Omron CX-Programmer project NewProject (CX-Programmer 9.50)

# PLC NewPLC1: CJ2M CPU35
I/O table (CPU CJ2M-CPU35): rack 0 slot 0 CJ1W-SCU41-V1; rack 0 slot 1 CJ1W-ID211; rack 0 slot 2 CJ1W-ID211; rack 0 slot 3 CJ1W-OC211; rack 0 slot 11 CJ2M-EIP21

## Global symbols (name address type ; comment)
0.00 BOOL  ; st
0.01 BOOL  ; sensor1
0.03 BOOL  ; metal detector
0.05 BOOL  ; sensor3
0.07 BOOL  ; sensor C4_R
0.09 BOOL  ; sensor C4_F
1.01 BOOL  ; sensor1
1.03 BOOL  ; SensorB2
1.05 BOOL  ; sensorP2_3
20.00 BOOL  ; st
20.01 BOOL  ; CR2
2.00 BOOL  ; e
2.01 BOOL  ; CR1
2.02 BOOL  ; pin28
2.03 BOOL  ; pin30
2.04 BOOL  ; pin36
2.05 BOOL  ; pin32
2.07 BOOL  ; gripper
2.09 BOOL  ; CR2
2.11 BOOL  ; CR1
2.13 BOOL  ; CR2_F
2.15 BOOL  ; CR2_R
3.00 BOOL  ; CR1
3.01 BOOL  ; CR2
T0004 BOOL  ; $?St$Bk?_#[5] / $?St$Bk?_#[5]
W0.00 BOOL  ; CR1
W0.01 BOOL  ; CR2
W0.02 BOOL  ; Continue
W0.03 BOOL  ; M1_forward
W0.04 BOOL  ; M1_reverse
W0.05 BOOL  ; M2_right
W0.06 BOOL  ; M2_left
W0.07 BOOL  ; arm_open
W0.08 BOOL  ; Continue process
W0.09 BOOL  ; stop
W0.10 BOOL  ; Start
W0.11 BOOL  ; Start
W0.12 BOOL  ; stop_button
W0.13 BOOL  ; stop
W0.14 BOOL  ; reset_button
W0.15 BOOL  ; cmd_Reset
W13.00 BOOL  ; Continue
W19.00 BOOL  ; btn_VB
W20.00 BOOL  ; btn_CX
W21.00 BOOL  ; Choose VB
W22.00 BOOL  ; Choose CX
W23.00 BOOL  ; status_VB
W24.00 BOOL  ; status_VB
W25.00 BOOL  ; status_CX
W2.00 BOOL  ; metal detect
W3.00 BOOL  ; destroy selfhold
W4.00 BOOL  ; the end of process_got 2 pcs
W6.00 BOOL  ; Reset W5

## Program NewProgram1 (cyclic task 0)
Local symbols
W INT
s UINT

### Section Section1

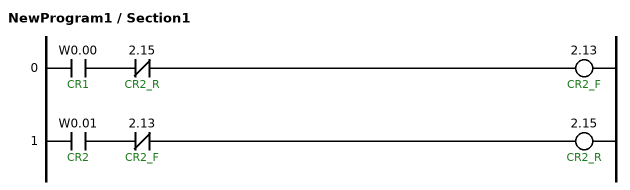
; rung 0
LD W0.00  ; CR1
ANDNOT 2.15  ; CR2_R
OUT 2.13  ; CR2_F
; rung 1
LD W0.01  ; CR2
ANDNOT 2.13  ; CR2_F
OUT 2.15  ; CR2_R

### Section state_transition

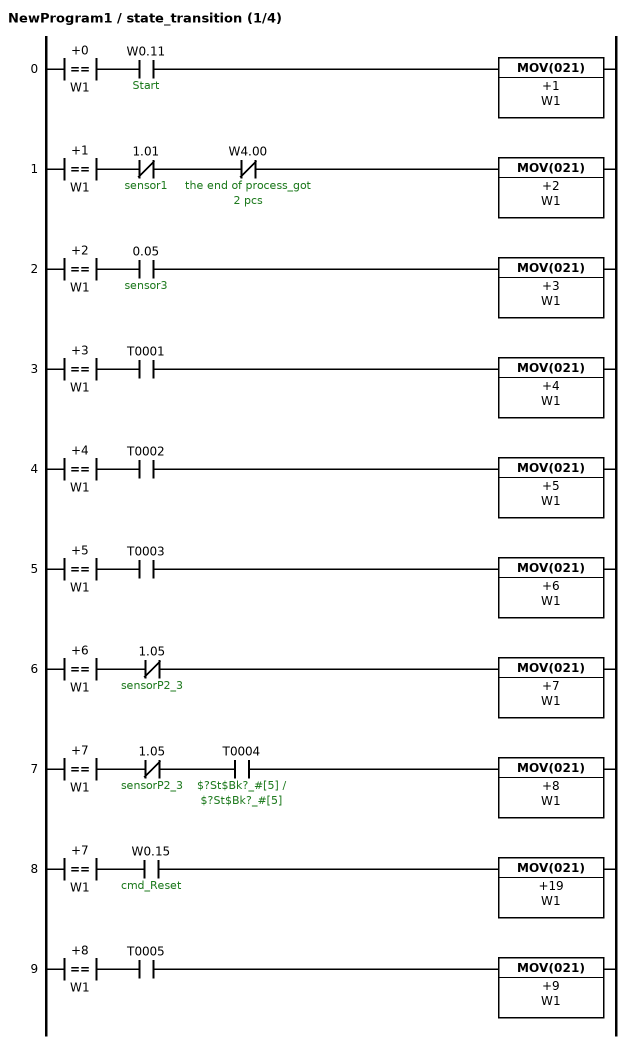
; rung 0
LD=S(302) +0 W1
AND W0.11  ; Start
MOV(021) +1 W1
; rung 1
LD=S(302) +1 W1
ANDNOT 1.01  ; sensor1
ANDNOT W4.00  ; the end of process_got 2 pcs
MOV(021) +2 W1
; rung 2
LD=S(302) +2 W1
AND 0.05  ; sensor3
MOV(021) +3 W1
; rung 3
LD=S(302) +3 W1
AND T0001
MOV(021) +4 W1
; rung 4
LD=S(302) +4 W1
AND T0002
MOV(021) +5 W1
; rung 5
LD=S(302) +5 W1
AND T0003
MOV(021) +6 W1
; rung 6
LD=S(302) +6 W1
ANDNOT 1.05  ; sensorP2_3
MOV(021) +7 W1
; rung 7
LD=S(302) +7 W1
ANDNOT 1.05  ; sensorP2_3
AND T0004  ; $?St$Bk?_#[5] / $?St$Bk?_#[5]
MOV(021) +8 W1
; rung 8
LD=S(302) +7 W1
AND W0.15  ; cmd_Reset
MOV(021) +19 W1
; rung 9
LD=S(302) +8 W1
AND T0005
MOV(021) +9 W1

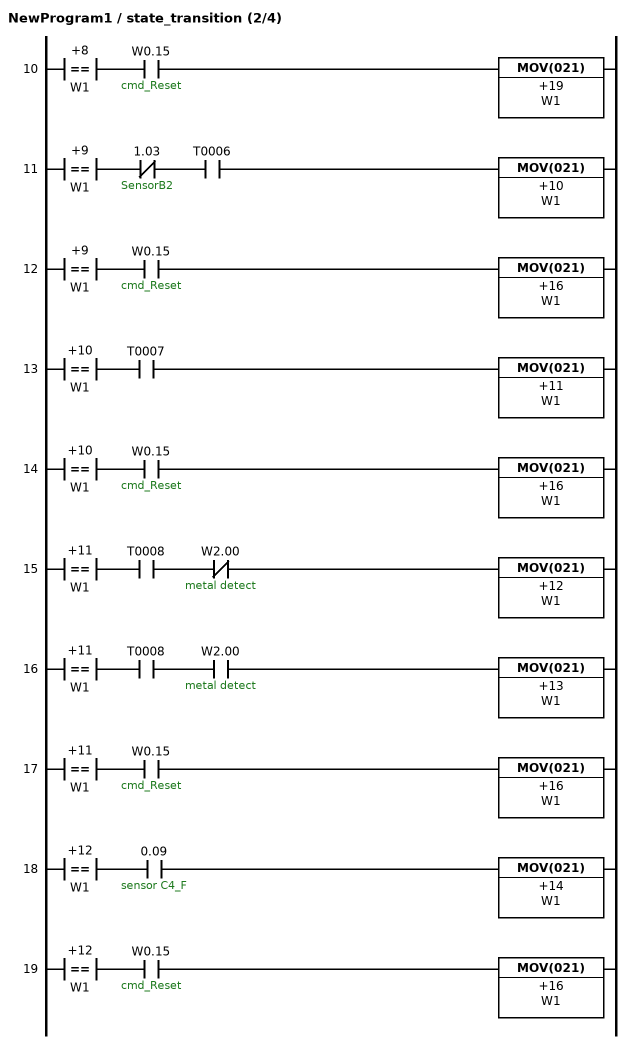
; rung 10
LD=S(302) +8 W1
AND W0.15  ; cmd_Reset
MOV(021) +19 W1
; rung 11
LD=S(302) +9 W1
ANDNOT 1.03  ; SensorB2
AND T0006
MOV(021) +10 W1
; rung 12
LD=S(302) +9 W1
AND W0.15  ; cmd_Reset
MOV(021) +16 W1
; rung 13
LD=S(302) +10 W1
AND T0007
MOV(021) +11 W1
; rung 14
LD=S(302) +10 W1
AND W0.15  ; cmd_Reset
MOV(021) +16 W1
; rung 15
LD=S(302) +11 W1
AND T0008
ANDNOT W2.00  ; metal detect
MOV(021) +12 W1
; rung 16
LD=S(302) +11 W1
AND T0008
AND W2.00  ; metal detect
MOV(021) +13 W1
; rung 17
LD=S(302) +11 W1
AND W0.15  ; cmd_Reset
MOV(021) +16 W1
; rung 18
LD=S(302) +12 W1
AND 0.09  ; sensor C4_F
MOV(021) +14 W1
; rung 19
LD=S(302) +12 W1
AND W0.15  ; cmd_Reset
MOV(021) +16 W1

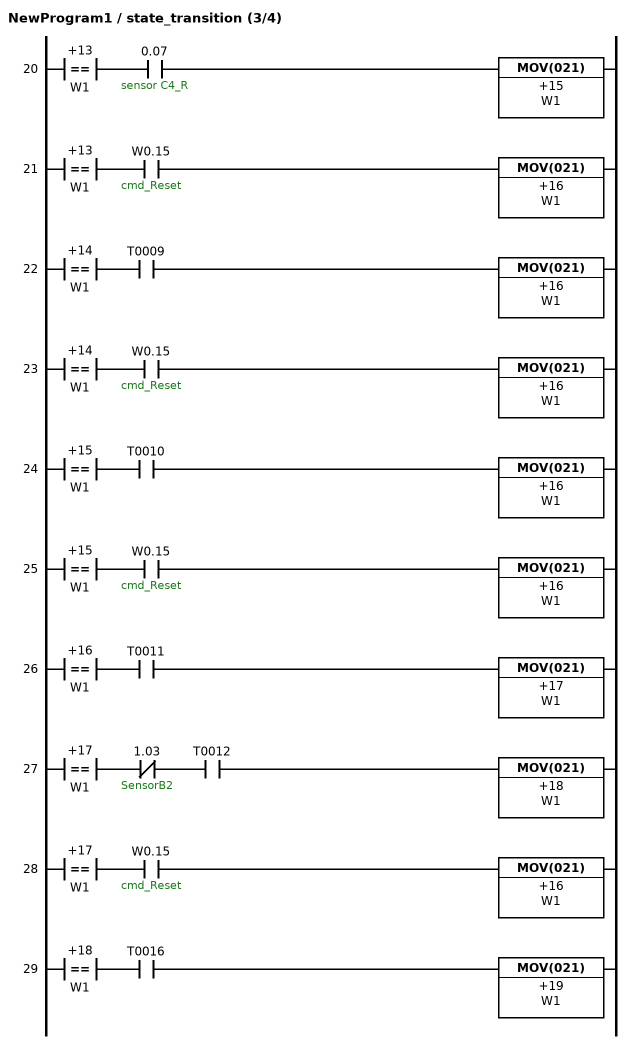
; rung 20
LD=S(302) +13 W1
AND 0.07  ; sensor C4_R
MOV(021) +15 W1
; rung 21
LD=S(302) +13 W1
AND W0.15  ; cmd_Reset
MOV(021) +16 W1
; rung 22
LD=S(302) +14 W1
AND T0009
MOV(021) +16 W1
; rung 23
LD=S(302) +14 W1
AND W0.15  ; cmd_Reset
MOV(021) +16 W1
; rung 24
LD=S(302) +15 W1
AND T0010
MOV(021) +16 W1
; rung 25
LD=S(302) +15 W1
AND W0.15  ; cmd_Reset
MOV(021) +16 W1
; rung 26
LD=S(302) +16 W1
AND T0011
MOV(021) +17 W1
; rung 27
LD=S(302) +17 W1
ANDNOT 1.03  ; SensorB2
AND T0012
MOV(021) +18 W1
; rung 28
LD=S(302) +17 W1
AND W0.15  ; cmd_Reset
MOV(021) +16 W1
; rung 29
LD=S(302) +18 W1
AND T0016
MOV(021) +19 W1

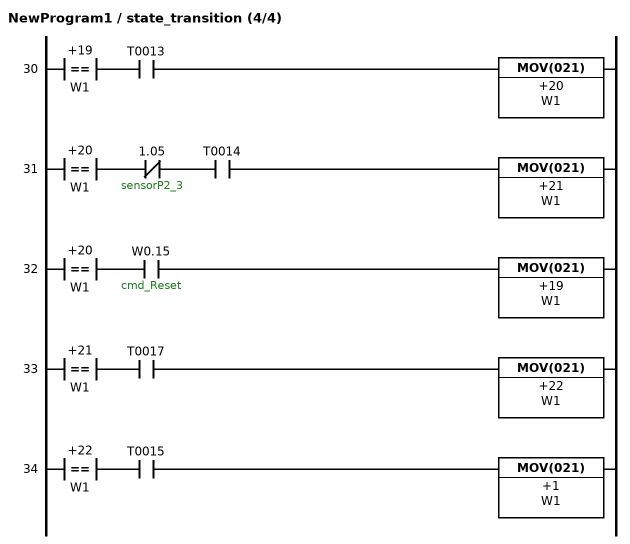
; rung 30
LD=S(302) +19 W1
AND T0013
MOV(021) +20 W1
; rung 31
LD=S(302) +20 W1
ANDNOT 1.05  ; sensorP2_3
AND T0014
MOV(021) +21 W1
; rung 32
LD=S(302) +20 W1
AND W0.15  ; cmd_Reset
MOV(021) +19 W1
; rung 33
LD=S(302) +21 W1
AND T0017
MOV(021) +22 W1
; rung 34
LD=S(302) +22 W1
AND T0015
MOV(021) +1 W1

### Section output_transition

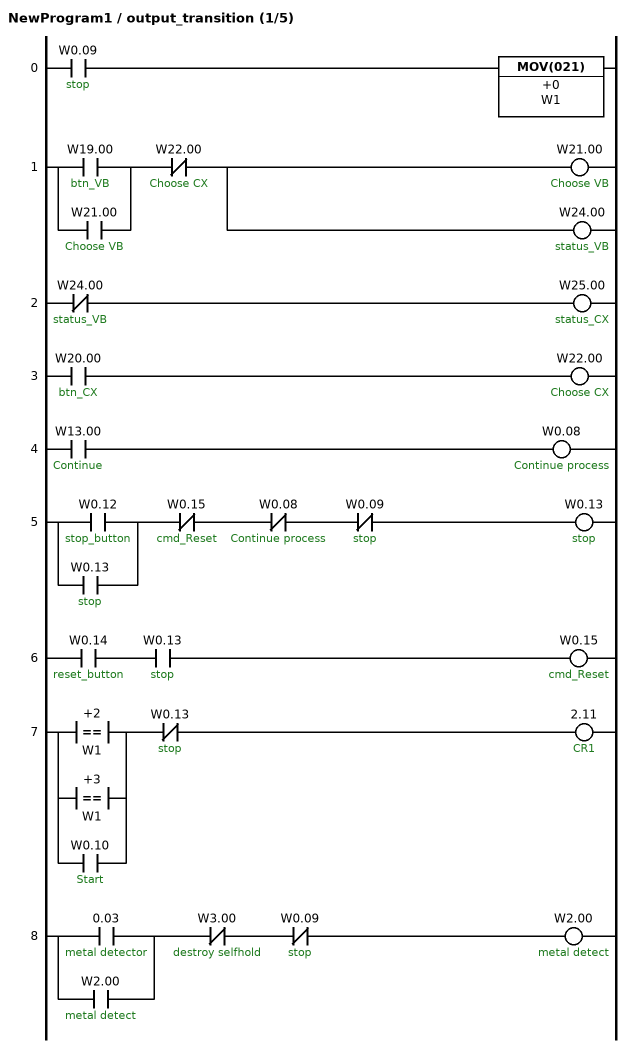
; rung 0
LD W0.09  ; stop
MOV(021) +0 W1
; rung 1
LD W19.00  ; btn_VB
OR W21.00  ; Choose VB
ANDNOT W22.00  ; Choose CX
OUT W21.00  ; Choose VB
OUT W24.00  ; status_VB
; rung 2
LDNOT W24.00  ; status_VB
OUT W25.00  ; status_CX
; rung 3
LD W20.00  ; btn_CX
OUT W22.00  ; Choose CX
; rung 4
LD W13.00  ; Continue
OUT W0.08  ; Continue process
; rung 5
LD W0.12  ; stop_button
OR W0.13  ; stop
ANDNOT W0.15  ; cmd_Reset
ANDNOT W0.08  ; Continue process
ANDNOT W0.09  ; stop
OUT W0.13  ; stop
; rung 6
LD W0.14  ; reset_button
AND W0.13  ; stop
OUT W0.15  ; cmd_Reset
; rung 7
LD=S(302) +2 W1
OR=S(302) +3 W1
OR W0.10  ; Start
ANDNOT W0.13  ; stop
OUT 2.11  ; CR1
; rung 8
LD 0.03  ; metal detector
OR W2.00  ; metal detect
ANDNOT W3.00  ; destroy selfhold
ANDNOT W0.09  ; stop
OUT W2.00  ; metal detect

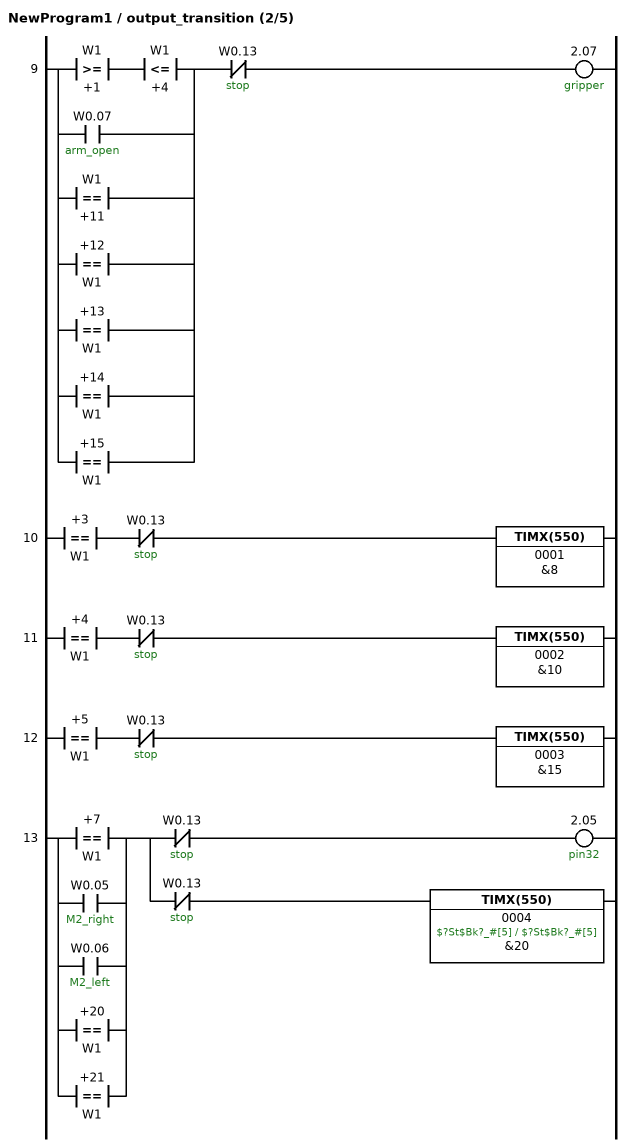
; rung 9
LD>=S(327) W1 +1
AND<=S(317) W1 +4
OR W0.07  ; arm_open
OR=S(302) W1 +11
OR=S(302) +12 W1
OR=S(302) +13 W1
OR=S(302) +14 W1
OR=S(302) +15 W1
ANDNOT W0.13  ; stop
OUT 2.07  ; gripper
; rung 10
LD=S(302) +3 W1
ANDNOT W0.13  ; stop
TIMX(550) 0001 &8
; rung 11
LD=S(302) +4 W1
ANDNOT W0.13  ; stop
TIMX(550) 0002 &10
; rung 12
LD=S(302) +5 W1
ANDNOT W0.13  ; stop
TIMX(550) 0003 &15
; rung 13
LD=S(302) +7 W1
OR W0.05  ; M2_right
OR W0.06  ; M2_left
OR=S(302) +20 W1
OR=S(302) +21 W1
OUT TR0
ANDNOT W0.13  ; stop
OUT 2.05  ; pin32
LD TR0
ANDNOT W0.13  ; stop
TIMX(550) 0004 &20  ; $?St$Bk?_#[5] / $?St$Bk?_#[5]

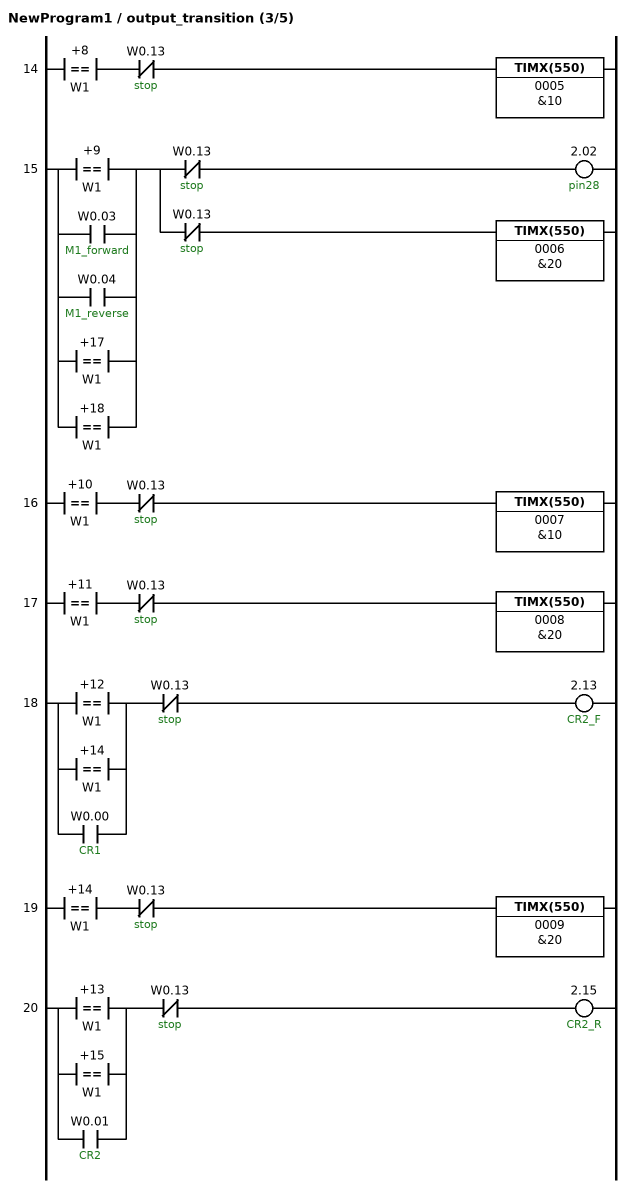
; rung 14
LD=S(302) +8 W1
ANDNOT W0.13  ; stop
TIMX(550) 0005 &10
; rung 15
LD=S(302) +9 W1
OR W0.03  ; M1_forward
OR W0.04  ; M1_reverse
OR=S(302) +17 W1
OR=S(302) +18 W1
OUT TR0
ANDNOT W0.13  ; stop
OUT 2.02  ; pin28
LD TR0
ANDNOT W0.13  ; stop
TIMX(550) 0006 &20
; rung 16
LD=S(302) +10 W1
ANDNOT W0.13  ; stop
TIMX(550) 0007 &10
; rung 17
LD=S(302) +11 W1
ANDNOT W0.13  ; stop
TIMX(550) 0008 &20
; rung 18
LD=S(302) +12 W1
OR=S(302) +14 W1
OR W0.00  ; CR1
ANDNOT W0.13  ; stop
OUT 2.13  ; CR2_F
; rung 19
LD=S(302) +14 W1
ANDNOT W0.13  ; stop
TIMX(550) 0009 &20
; rung 20
LD=S(302) +13 W1
OR=S(302) +15 W1
OR W0.01  ; CR2
ANDNOT W0.13  ; stop
OUT 2.15  ; CR2_R

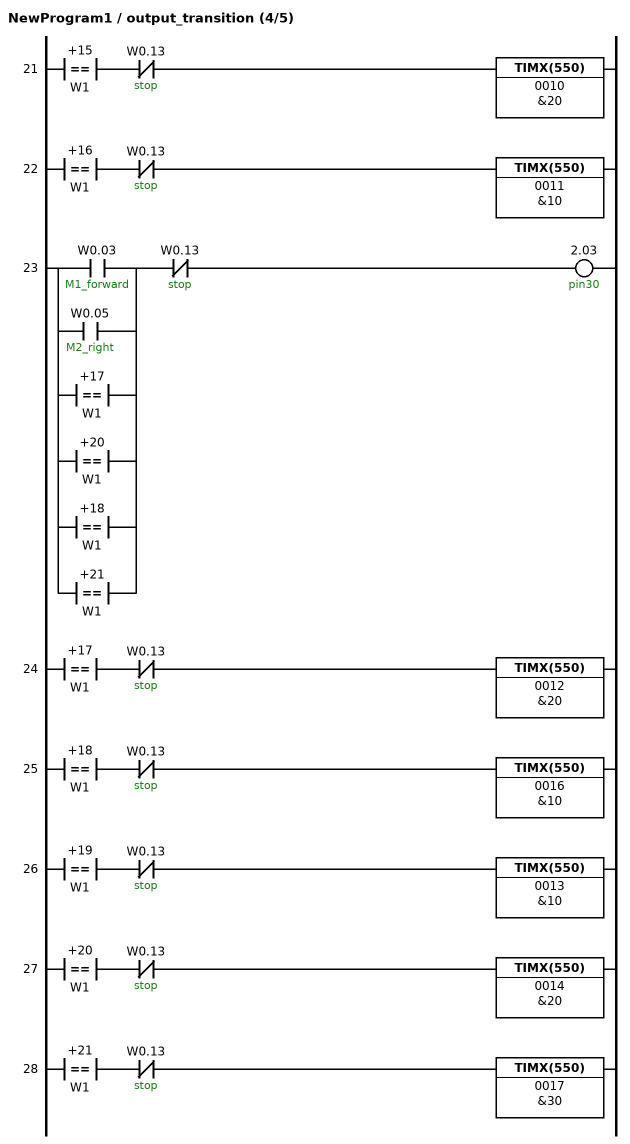
; rung 21
LD=S(302) +15 W1
ANDNOT W0.13  ; stop
TIMX(550) 0010 &20
; rung 22
LD=S(302) +16 W1
ANDNOT W0.13  ; stop
TIMX(550) 0011 &10
; rung 23
LD W0.03  ; M1_forward
OR W0.05  ; M2_right
OR=S(302) +17 W1
OR=S(302) +20 W1
OR=S(302) +18 W1
OR=S(302) +21 W1
ANDNOT W0.13  ; stop
OUT 2.03  ; pin30
; rung 24
LD=S(302) +17 W1
ANDNOT W0.13  ; stop
TIMX(550) 0012 &20
; rung 25
LD=S(302) +18 W1
ANDNOT W0.13  ; stop
TIMX(550) 0016 &10
; rung 26
LD=S(302) +19 W1
ANDNOT W0.13  ; stop
TIMX(550) 0013 &10
; rung 27
LD=S(302) +20 W1
ANDNOT W0.13  ; stop
TIMX(550) 0014 &20
; rung 28
LD=S(302) +21 W1
ANDNOT W0.13  ; stop
TIMX(550) 0017 &30

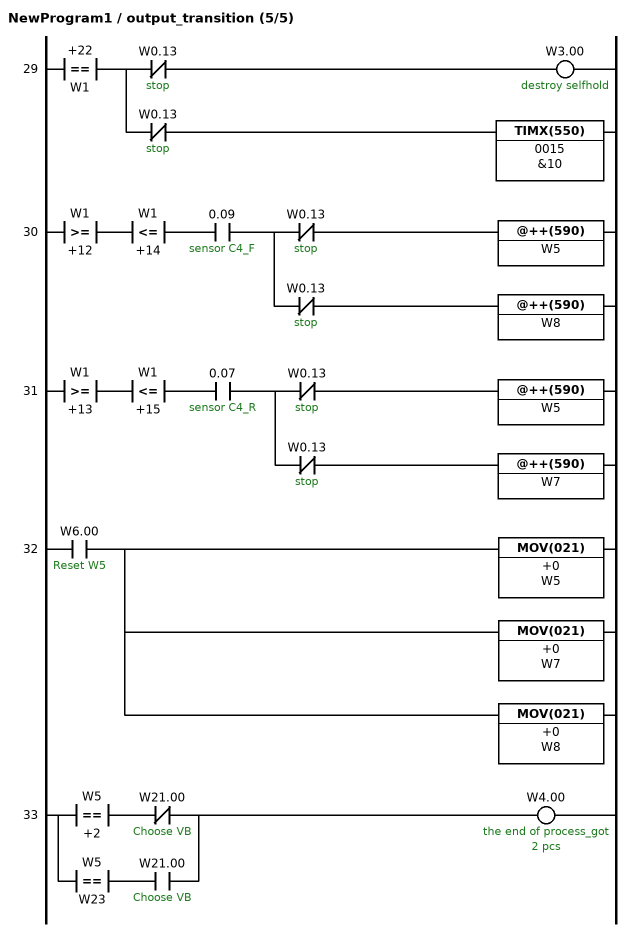
; rung 29
LD=S(302) +22 W1
OUT TR0
ANDNOT W0.13  ; stop
OUT W3.00  ; destroy selfhold
LD TR0
ANDNOT W0.13  ; stop
TIMX(550) 0015 &10
; rung 30
LD>=S(327) W1 +12
AND<=S(317) W1 +14
AND 0.09  ; sensor C4_F
OUT TR0
ANDNOT W0.13  ; stop
@++(590) W5
LD TR0
ANDNOT W0.13  ; stop
@++(590) W8
; rung 31
LD>=S(327) W1 +13
AND<=S(317) W1 +15
AND 0.07  ; sensor C4_R
OUT TR0
ANDNOT W0.13  ; stop
@++(590) W5
LD TR0
ANDNOT W0.13  ; stop
@++(590) W7
; rung 32
LD W6.00  ; Reset W5
MOV(021) +0 W5
MOV(021) +0 W7
MOV(021) +0 W8
; rung 33
LD=S(302) W5 +2
ANDNOT W21.00  ; Choose VB
LD=S(302) W5 W23
AND W21.00  ; Choose VB
ORLD
OUT W4.00  ; the end of process_got 2 pcs

### Section END
; rung 0
END(001)